(* PLC project Cell Example , CTH FIX1 1.0, author CTH SS2 *)
(* stored: companyURL www.chalmers.se, creationDateTime 2008-03-19T20:31:26, version 1.0, modificationDateTime 2008-04-25T16:51:04, organization SS2, language en-US *)

TYPE BinaryPositions : ();
END_TYPE

FUNCTION ADD_E : INT
  VAR_INPUT
    Enable : BOOL := FALSE;
    IN1 : INT := 0;
    IN2 : INT := 0;
  END_VAR
  VAR_OUTPUT
    EnableO : BOOL := FALSE;
  END_VAR

(* LD diagram, written out as Structured Text *)
END_FUNCTION

FUNCTION DEC_E : INT
  VAR_INPUT
    Enable : BOOL;
  END_VAR
  VAR_OUTPUT
    EnableO : BOOL;
  END_VAR

(* LD diagram, written out as Structured Text *)
END_FUNCTION

FUNCTION MOVE_E : STRING
  VAR_INPUT
    Enable : BOOL := FALSE;
    IN : STRING;
  END_VAR
  VAR_OUTPUT
    EnableO : BOOL := FALSE;
  END_VAR

(* LD diagram, written out as Structured Text *)
END_FUNCTION

FUNCTION_BLOCK RAC
  VAR_INPUT
    IN1 : BOOL := FALSE;
  END_VAR
  VAR_OUTPUT
    OUT : BOOL := FALSE;
  END_VAR
  VAR_INPUT
    IN2 : BOOL := TRUE;
  END_VAR
  VAR
    Var3 : BOOL := TRUE;
    IN4 : INT := 5;
  END_VAR
  VAR_OUTPUT
    State : STRING := 'Undefined';
  END_VAR
  VAR
    timer : TON;
    passedTime : TIME := 20;
  END_VAR
  VAR  (* added by the conversion: wires and edge detectors of the diagram *)
    _ADD_E24_ : ANY;
    _ADD_E24_OUT : INT;
    _MOVE_E26_ : ANY;
    _MOVE_E26_OUT : STRING;
    _DEC_E34_ : ANY;
    _DEC_E34_OUT : INT;
  END_VAR

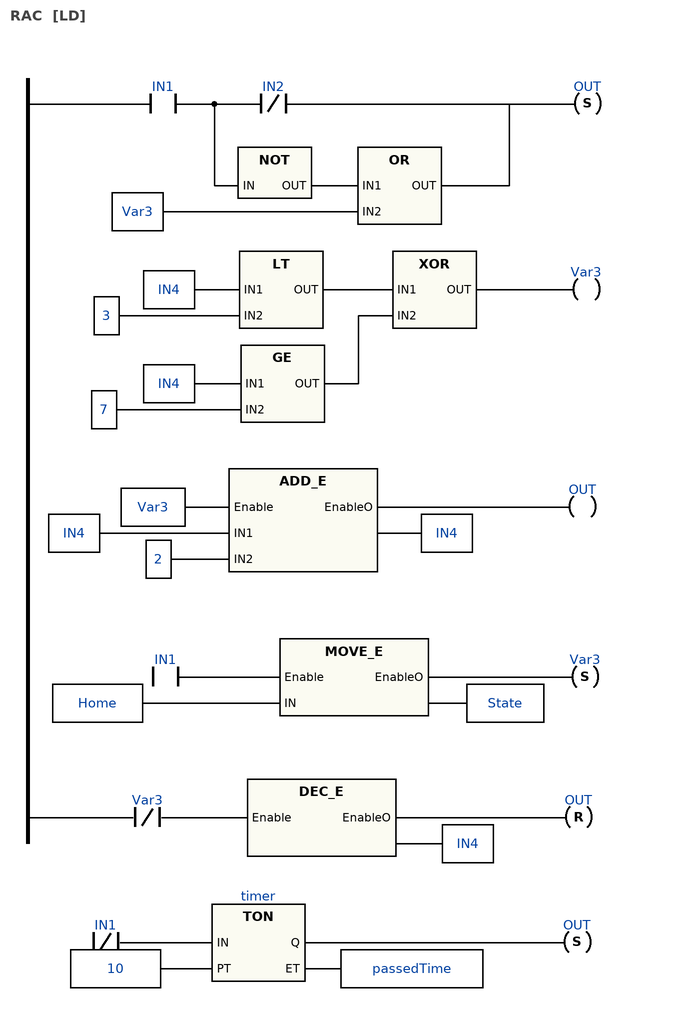
(* LD diagram, written out as Structured Text *)
IF IN1 AND NOT IN2 OR NOT IN1 OR Var3 THEN OUT := TRUE; END_IF;
Var3 := IN4 < 3 XOR IN4 >= 7;
_ADD_E24_OUT := ADD_E(Enable := Var3, IN1 := IN4, IN2 := 2,  => _ADD_E24_);
OUT := _ADD_E24_OUT;
IN4 := _ADD_E24_OUT;
_MOVE_E26_OUT := MOVE_E(Enable := IN1, IN := Home,  => _MOVE_E26_);
IF _MOVE_E26_OUT THEN Var3 := TRUE; END_IF;
State := _MOVE_E26_OUT;
_DEC_E34_OUT := DEC_E(Enable := NOT Var3,  => _DEC_E34_);
IF _DEC_E34_OUT THEN OUT := FALSE; END_IF;
IN4 := _DEC_E34_OUT;
timer(IN := NOT IN1, PT := 10);
IF timer.Q THEN OUT := TRUE; END_IF;
passedTime := timer.ET;
END_FUNCTION_BLOCK

CONFIGURATION ExampleCell
END_CONFIGURATION
